Universal Robots PolyScope program: Socket_example.urp

Program Socket_example (installation=default directory=/home/ur/ursim-current/programs createdIn=5.10.0.106288 lastSavedIn=5.10.0.106288 robotSerialNumber=20195599999)
Calibrated DH parameters: a=[0, -0.425, -0.3922, 0, 0, 0]; d=[0.1625, 0, 0, 0.1333, 0.0997, 0.0996]; alpha=[1.570796, 0, 0, 1.570796, -1.570796, 0]; deltaTheta=[0, 0, 0, 0, 0, 0]
BeforeStart
  Script: socket_close()
  conn := False
  targetPos := p[0,0,0,0,0,0]
  count := 0
  Loop While (checkContinuously=false) expression=conn≟ False
    conn := socket_open("192.168.56.102", 50000)
    Wait Sleep waitTime=0.01
Robot Program (runOnlyOnce=true)
  MoveJ speed 60 deg/s, acceleration 80 deg/s^2 (useActiveTCP=true) feature=Base
    Waypoint Start: TCP in base x=-143.969 y=-435.62 z=202.03 mm, rx=-0.0012 ry=3.1163 rz=0.0389 rad; joints [-91.713, -98.956, -126.223, -46.295, 91.392, -1.776] deg
  Script: socket_send_string("get pose")
  response := socket_read_ascii_float(6)
  Loop While (checkContinuously=false) expression=response[0]≠6
    Wait Sleep waitTime=0.01
    response := socket_read_ascii_float(6)
  Loop While (checkContinuously=false) expression=count<6
    Script: targetPos[count]=response[count+1]
    count := count+1
  MoveJ speed 60 deg/s, acceleration 80 deg/s^2 (useActiveTCP=true) feature=Base
    Waypoint Waypoint (Variable): variable=targetPos
  Script: socket_close()
